TYPE T_TriggerControlBits :
STRUCT
  Enable        : BIT;
  Init          : BIT;
  NoFeedback    : BIT;
{attribute 'hide'} 
  b3            : BIT;
{attribute 'hide'} 
  b4            : BIT;
{attribute 'hide'} 
  b5            : BIT;
{attribute 'hide'} 
  b6            : BIT;
{attribute 'hide'} 
  b7            : BIT;
END_STRUCT
END_TYPE

(* stored: Version 1.1.0.1
   DUT T_TriggerControlBits: Id {7eb5c1cb-9de2-4b09-8f3d-741a7cef6cdf} *)
